// TIA Portal V18 export
// export: Created 2026-06-03T07:11:57.0146873Z, ExportSetting WithDefaults, DisplayName Totally Integrated Automation Portal, DisplayVersion V18, DisplayName TIA Portal Openness, DisplayVersion V18, DisplayName TIA Portal Version Control Interface, DisplayVersion V18, DisplayName STEP 7 Professional, DisplayVersion V18, DisplayName STEP 7 Safety, DisplayVersion V18, DisplayName WinCC Professional, DisplayVersion V18
Screen "04_Trend"  800x600, Number=4
  ScreenLayer 
    GraphicView "Graphic view_1" at 0,0 size 800x600  Picture=Màn Trend
    Button "Button_1" at 27,538 size 107x46  Mode=Text, TextOff="TỔNG QUAN", TextOn="Text"
      on Click: ActivateScreen(Screen name := 01_Tong_Quan, Object number := 0)
    Button "Button_2" at 153,538 size 107x46  Mode=Text, TextOff="VẬN HÀNH", TextOn="Text"
      on Click: ActivateScreen(Screen name := 02_Van_Hanh, Object number := 0)
    Button "Button_3" at 281,538 size 107x46  Mode=Text, TextOff="PID MỨC", TextOn="Text"
      on Click: ActivateScreen(Screen name := 03_PID_Muc_Nuoc, Object number := 0)
    Button "Button_5" at 537,537 size 107x46  Mode=Text, TextOff="CẢNH BÁO", TextOn="Text"
      on Click: ActivateScreen(Screen name := 05_Canh_Bao_IO, Object number := 0)
    TextField "Text field_1" at 245,13 size 251x31  Text="MÀN HÌNH 4- TRENDS"
    Circle "Circle_3" at 677,3 size 39x39
      RangeAppearanceAnimation "RangeAppearanceAnimation"
        tag bSystemRun
        0..0: back #d9d9d9, fore #181c31
        1..1: back #00ff00, fore #181c31
    Circle "Circle_2" at 718,3 size 39x39
      RangeAppearanceAnimation "RangeAppearanceAnimation"
        tag Loi_He_Thong
        0..0: back #d9d9d9, fore #181c31
        1..1: back #ff0000, fore #181c31
    Circle "Circle_1" at 759,3 size 39x39
      RangeAppearanceAnimation "RangeAppearanceAnimation"
        tag bCheDoMoPhong
        0..0: back #d9d9d9, fore #181c31
        1..1: back #0000ff, fore #181c31
    TextField "Text field_2" at 679,40 size 34x22  Text="Run"
    TextField "Text field_3" at 717,40 size 43x22  Text="Fault"
    TextField "Text field_4" at 760,40 size 33x22  Text="Sim"
    Rectangle "Rectangle_8" at 405,536 size 114x52
    Button "Button_4" at 409,539 size 107x46  Mode=Text, TextOff="TREND", TextOn="Text"
      on Click: ActivateScreen(Screen name := , Object number := 0)
    Button "Button_6" at 729,559 size 65x30  Mode=Text, TextOff="EXIT", TextOn="Text"
      on Click: StopRuntime(Mode := 0)
    Button "Button_7" at 32,390 size 116x73  Mode=Text, TextOff="MỨC NƯỚC PV", TextOn="Text"
      on Click: Toggle_PV()
    Button "Button_8" at 186,390 size 116x73  Mode=Text, TextOff="MỨC NƯỚC SP", TextOn="Text"
      on Click: Toggle_PV()
    Button "Button_9" at 340,390 size 116x73  Mode=Text, TextOff="ĐỘ MỞ VAN OP", TextOn="Text"
      on Click: Toggle_OP()
    Button "Button_10" at 498,390 size 116x73  Mode=Text, TextOff="NHIỆT ĐỘ BỒN", TextOn="Text"
      on Click: Toggle_Temp()
    Button "Button_11" at 655,390 size 116x73  Mode=Text, TextOff="ÁP SUẤT LÒ HƠI", TextOn="Text"
      on Click: Toggle_Press()
    Rectangle "Rectangle_1" at 671,72 size 113x47
    IOField "I/O field_3" at 693,95 size 49x24  DataFormat=Decimal, FormatPattern=9.9, Mode=Output
      ProcessValue := Muc_Nuoc_PV
    TextField "Text field_18" at 736,96 size 17x22  Text="m"
    Rectangle "Rectangle_2" at 671,127 size 112x47
    IOField "I/O field_4" at 693,148 size 49x24  DataFormat=Decimal, FormatPattern=9.9, Mode=Output
      ProcessValue := Muc_Nuoc_SP
    TextField "Text field_17" at 736,149 size 17x22  Text="m"
    Rectangle "Rectangle_3" at 672,72 size 112x22
    TextField "Text field_14" at 673,74 size 110x19  Text="Mức nước thực tế"
    Rectangle "Rectangle_4" at 671,127 size 112x22
    TextField "Text field_15" at 673,128 size 107x19  Text="Mức nước cài đặt"
    Rectangle "Rectangle_5" at 671,183 size 112x47
    Rectangle "Rectangle_6" at 671,183 size 112x22
    TextField "Text field_5" at 681,185 size 84x19  Text="Độ mở van xả"
    IOField "I/O field_5" at 696,205 size 49x24  DataFormat=Decimal, FormatPattern=99.9, Mode=Output
      ProcessValue := Van_Xa_OP
    TextField "Text field_19" at 739,207 size 18x22  Text="%"
    Rectangle "Rectangle_7" at 671,241 size 112x47
    Rectangle "Rectangle_9" at 671,241 size 112x22
    TextField "Text field_6" at 687,244 size 75x19  Text="Nhiệt độ bồn"
    IOField "I/O field_1" at 696,263 size 49x24  DataFormat=Decimal, FormatPattern=99.9, Mode=Output
      ProcessValue := Nhiet_Do_PV
    TextField "Text field_21" at 738,265 size 23x22  Text="°C"
    Rectangle "Rectangle_10" at 671,301 size 112x47
    Rectangle "Rectangle_11" at 671,301 size 112x22
    TextField "Text field_7" at 695,303 size 61x19  Text="Áp suất lò"
    IOField "I/O field_2" at 693,324 size 49x24  DataFormat=Decimal, FormatPattern=99.9, Mode=Output
      ProcessValue := Ap_Suat_PV
    TextField "Text field_20" at 738,325 size 31x22  Text="Bar"
